// TIA Portal V19 export
FUNCTION "PNIO Node Diag State" : Void   // FC301, STL
TITLE = PNIO Node Diagnostic Error bits
{ S7_Optimized_Access := 'TRUE' }
// This function take a PNIO "module diagnostic result" word and outputs the active
//  
// bits. 
// Bit 1.0 = Node Failed
// Bit 1.1 = Module Fault
// Bit 1.2 = Maintenance Required
// stored: AutoNumber false
   VAR_INPUT
      nodeDiag : Int;
   END_VAR
   VAR_OUTPUT
      failed : Bool;
      moduleFault : Bool;
      maintenanceReq : Bool;
   END_VAR
BEGIN

NETWORK
TITLE = 
      A     #nodeDiag.%X1;
      =     #failed;
      A     #nodeDiag.%X4;
      =     #moduleFault;
      A     #nodeDiag.%X2;
      O     #nodeDiag.%X3;
      O     #nodeDiag.%X5;
      O     #nodeDiag.%X6;
      =     #maintenanceReq;

END_FUNCTION
